Yaskawa INFORM job: FRONT_SEARCH_180ST_5040_1.JBI

/JOB
//NAME FRONT_SEARCH_180ST_5040_1
///FOLDERNAME 02-SKRZYNIE_JOBS
//POS
///NPOS 44,44,0,3,0,0
///TOOL 0
///POSTYPE PULSE
///PULSE
C00000=0,-52280,40443,0,6876,0
C00001=90,-52869,30671,-35,13158,-11387
C00002=3,-35052,15441,1,18785,-31206
C00003=-69983,-39842,-15225,22698,60757,-54805
C00004=-95672,-18401,-524,43648,77081,-65694
C00005=-95672,-18401,-524,43648,77081,-65694
C00006=-66488,-10859,14335,53179,60119,-60859
C00007=-64335,-9865,15970,53979,58765,-60616
C00008=-62298,-8078,17660,53897,57781,-60133
C00009=-64335,-9865,15970,53979,58765,-60616
C00010=-60965,-12473,13602,54156,56779,-60101
C00011=-73399,577,26586,53509,63912,-62118
C00012=-73399,2178,31028,54225,62862,-62902
C00013=-73399,577,26586,53509,63912,-62118
C00014=-95672,-18401,-524,43648,77081,-65694
C00015=-95672,-18401,-524,43648,77081,-65694
C00016=-78752,-37675,-14240,25444,65481,-57695
C00017=-81739,-44645,-17805,23160,61789,-58708
C00018=-60964,-50253,-20349,19915,49744,-52813
///LIMIT ON
C00019=252,-53930,13084,-98,24463,-31882
///LIMIT OFF
C00020=0,-52280,40443,0,6876,0
C00021=0,-52280,40443,0,6876,0
///LIMIT ON
C00022=-252,-53930,13084,98,24463,31882
///LIMIT OFF
C00023=63842,-57146,-8568,-22669,38929,56818
C00024=57252,-42862,-8372,-20543,46199,52542
C00025=95672,-18401,-524,-43648,77081,65694
C00026=95672,-18401,-524,-43648,77081,65694
C00027=67931,-13462,11045,-52218,61046,61006
C00028=62394,-11410,14553,-54081,57623,60319
C00029=60703,-9918,15919,-53986,56824,59903
C00030=62394,-11410,14553,-54081,57623,60319
C00031=58733,-14007,12260,-54261,55457,59764
C00032=62394,-11410,14553,-54081,57623,60319
C00033=69392,-7516,18202,-53778,61595,61493
C00034=69392,-4008,27735,-55517,59418,63215
C00035=66736,-2123,29102,-55452,58266,62512
C00036=66736,-2869,27102,-55056,58712,62144
C00037=68586,-4452,25471,-54998,59658,62519
C00038=62394,-11410,14553,-54081,57623,60319
C00039=95672,-18401,-524,-43648,77081,65694
C00040=100154,-19751,-1600,-43338,78981,66779
C00041=50663,-34953,14820,-22623,45539,36921
C00042=25336,-44267,23454,-10793,27790,20731
C00043=0,-52280,40443,0,6876,0
BC00000=837049
BC00001=850281
BC00002=878680
BC00003=890984
BC00004=908397
BC00005=941160
BC00006=941160
BC00007=941160
BC00008=941160
BC00009=941160
BC00010=941160
BC00011=941160
BC00012=941160
BC00013=941160
BC00014=941160
BC00015=908397
BC00016=893750
BC00017=890385
BC00018=884436
BC00019=813034
BC00020=801491
BC00021=801491
BC00022=813034
BC00023=862329
BC00024=879547
BC00025=908397
BC00026=941160
BC00027=941160
BC00028=941160
BC00029=941160
BC00030=941160
BC00031=941160
BC00032=941160
BC00033=941160
BC00034=941160
BC00035=941160
BC00036=941160
BC00037=941160
BC00038=941160
BC00039=941160
BC00040=908397
BC00041=860901
BC00042=834175
BC00043=801491
///POSTYPE BASE
///RECTAN
///RCONF 1,0,0,0,0,0,0,0,0,0,0,0,0,0,0,0,0,0,0,0,0,0,0,0
P00006=0.000,0.000,0.000,0.0000,0.0000,0.0000
///RCONF 0,0,0,0,0,0,0,0,0,0,0,0,0,0,0,0,0,0,0,0,0,0,0,0
P00400=5.920,-3.503,-0.024,0.0000,0.0000,0.0000
P00401=3.430,-0.021,1.131,0.0000,0.0000,0.0000
//INST
///DATE 2024/05/14 12:08
///ATTR SC,RW
///GROUP1 RB1,BS1
NOP
MOVJ C00000 BC00000 VJ=30.00
MOVJ C00001 BC00001 VJ=30.00
MOVJ C00002 BC00002 VJ=10.00
MOVJ C00003 BC00003 VJ=10.00
MOVJ C00004 BC00004 VJ=10.00
MOVJ C00005 BC00005 VJ=25.00
'------------------------
'W32
'------------------------
MOVL C00006 BC00006 V=500.0
MOVL C00007 BC00007 V=66.7 PL=0
REFP 3 C00008 BC00008
CALL JOB:SEARCH-R1
SET P0400 P0006
SFTON P0400
MOVL C00009 BC00009 V=66.7 PL=0
REFP 3 C00010 BC00010
CALL JOB:SEARCH-R1
SET P0400 P0006
SFTON P0400
MOVL C00011 BC00011 V=66.7 PL=0
REFP 3 C00012 BC00012
CALL JOB:SEARCH-R1
SET P0400 P0006
SFTON P0400
MOVL C00013 BC00013 V=66.7 PL=0
SFTOF
MOVJ C00014 BC00014 VJ=20.00
MOVJ C00015 BC00015 VJ=20.00
MOVJ C00016 BC00016 VJ=15.00
MOVJ C00017 BC00017 VJ=20.00
MOVJ C00018 BC00018 VJ=20.00
MOVJ C00019 BC00019 VJ=25.00
MOVJ C00020 BC00020 VJ=50.00
'TEST
'TEST
'TEST
'TEST
MOVJ C00021 BC00021 VJ=5.00
MOVJ C00022 BC00022 VJ=15.00
MOVJ C00023 BC00023 VJ=15.00
MOVJ C00024 BC00024 VJ=10.00 PL=0
MOVJ C00025 BC00025 VJ=10.00 PL=0
MOVJ C00026 BC00026 VJ=25.00
'------------------------
'W32
'------------------------
MOVL C00027 BC00027 V=500.0
MOVL C00028 BC00028 V=133.3 PL=0
REFP 3 C00029 BC00029
CALL JOB:SEARCH-R1
SET P0401 P0006
SFTON P0401
MOVL C00030 BC00030 V=66.7 PL=0
REFP 3 C00031 BC00031
CALL JOB:SEARCH-R1
SET P0401 P0006
SFTON P0401
MOVL C00032 BC00032 V=66.7
MOVL C00033 BC00033 V=133.3
MOVL C00034 BC00034 V=133.3
MOVL C00035 BC00035 V=66.7 PL=0
REFP 3 C00036 BC00036
CALL JOB:SEARCH-R1
SET P0401 P0006
SFTON P0401
MOVL C00037 BC00037 V=66.7
MOVL C00038 BC00038 V=66.7 PL=0
SFTOF
MOVJ C00039 BC00039 VJ=10.00
MOVJ C00040 BC00040 VJ=20.00 PL=0
MOVJ C00041 BC00041 VJ=10.00 PL=0
MOVJ C00042 BC00042 VJ=25.00
MOVJ C00043 BC00043 VJ=50.00
END
